(*
SPDX-FileCopyrightText: © 2026 Oleksandr Tiutyk <trofimich@gmail.com>
SPDX-License-Identifier: MIT
License: https://opensource.org/license/mit
*)

{attribute 'no_explicit_call' := 'do not call this function block directly'} 
{attribute 'enable_dynamic_creation'}
FUNCTION_BLOCK WaitAndPickActivity EXTENDS ExclusiveCompositeActivity IMPLEMENTS IWaitAndPickActivity
VAR
	{attribute 'OPC.UA.DA' := '0'}
	_ClassName : STRING := __POUNAME();

	{attribute 'OPC.UA.DA' := '0'}
	_BranchConditions : TOF_Collections.List<0>(0);

	{attribute 'OPC.UA.DA' := '0'}
	_BranchActivities : TOF_Collections.List<0>(0);
	
	{attribute 'OPC.UA.DA' := '0'}	
	_CurrentBranchIndex : DINT := -1;
END_VAR

METHOD AddBarnch : DINT
VAR_INPUT
	condition : ICondition;
	activity : IActivity;
END_VAR
VAR
	conditionNullExcxeption : TOF_Core.ArgumentNotSpecifiedException;
	activityNullExcxeption : TOF_Core.ArgumentNotSpecifiedException;
END_VAR
IF condition = 0  THEN
	activityNullExcxeption.Throw(NamespaceName, ClassName, __POUNAME(), __POSITION(), 'condition');
END_IF

IF activity = 0  THEN
	activityNullExcxeption.Throw(NamespaceName, ClassName, __POUNAME(), __POSITION(), 'activity');
END_IF

activity.ParentActivity := THIS^;

_BranchConditions.AppendGeneric(TOF_Core.GenericValueFactory.FromParts(TOF_Core.GENERIC_TYPE_CLASS.OBJECT, condition.SelfAddress, condition.SelfSize, TOF_Core.GENERIC_MEMORY_MANAGEMENT_BEHAVIOR.STORE_ORIGINAL_REFERENCE_AND_NOT_OWNS_MEMORY));

_BranchActivities.AppendGeneric(TOF_Core.GenericValueFactory.FromParts(TOF_Core.GENERIC_TYPE_CLASS.OBJECT, activity.SelfAddress, activity.SelfSize, TOF_Core.GENERIC_MEMORY_MANAGEMENT_BEHAVIOR.STORE_ORIGINAL_REFERENCE_AND_NOT_OWNS_MEMORY), index => AddBarnch);
END_METHOD

{attribute 'monitoring' := 'call'}
PROPERTY ClassName : REFERENCE TO STRING
GET
ClassName REF= _ClassName;
END_GET
END_PROPERTY

{attribute 'monitoring' := 'call'}
PROPERTY FINAL CurrentActivity : IActivity
GET
IF _BranchActivities.Length > 0 AND_THEN _CurrentBranchIndex >= 0 AND_THEN _CurrentBranchIndex < _BranchActivities.Length THEN
	__QUERYINTERFACE(_BranchActivities.Get(_CurrentBranchIndex).AsObject(), CurrentActivity);
END_IF
END_GET
END_PROPERTY

{attribute 'monitoring' := 'call'}
PROPERTY FINAL CurrentBranchIndex : DINT
GET
CurrentBranchIndex := _CurrentBranchIndex;
END_GET
END_PROPERTY

{attribute 'monitoring' := 'call'}
PROPERTY NamespaceName : REFERENCE TO STRING
GET
NamespaceName REF= CurrentNamespace.Name;
END_GET
END_PROPERTY

METHOD PROTECTED OnCancelling 
VAR_INPUT
	start : BOOL;
END_VAR
VAR_OUTPUT
	cancelled : BOOL;
END_VAR
VAR
	activity : IActivity;
END_VAR
END_METHOD

METHOD PROTECTED OnRunning : ACTIVITY_RUNNING_STATE
VAR_INPUT
	startRunning : BOOL;
	startResuming : BOOL;
END_VAR
VAR_OUTPUT
	haltReason : WSTRING(255);
END_VAR
VAR
	activity : IActivity;
	
	currentActivityNullException : TOF_Core.NullReferenceException;
END_VAR
IF _BranchConditions.Length < 1 THEN
	OnRunning := ACTIVITY_RUNNING_STATE.WORK_COMPLETED;
	RETURN;
END_IF

IF startRunning THEN
	_CurrentBranchIndex := -1;
END_IF

IF _CurrentBranchIndex < 0 THEN
	_CurrentBranchIndex := tryPickBranch();
END_IF

IF _CurrentBranchIndex < 0 THEN
	RETURN;
END_IF

activity := CurrentActivity;

IF activity = 0 THEN
	currentActivityNullException.Throw(NamespaceName, ClassName, __POUNAME(), __POSITION(), 'CurrentActivity');
END_IF

IF startRunning OR_ELSE startResuming OR_ELSE NOT activity.Busy THEN
	activity.RequestStart();
ELSE
	activity.Execute();
END_IF

OnRunning := GetActivityRunningStateByNestedActivityState(activity.State);
END_METHOD

METHOD PROTECTED OnStopping : ACTIVITY_STOPPING_STATE
VAR_INPUT
	startCancelling : BOOL;
	startSuspending : BOOL;
END_VAR
VAR_OUTPUT
	haltReason : WSTRING(255);
END_VAR
VAR
	activity : IActivity;
END_VAR
IF _BranchConditions.Length < 1 THEN
	OnStopping := ACTIVITY_STOPPING_STATE.WORK_COMPLETED;
	RETURN;
END_IF

activity := CurrentActivity;

IF activity = 0 THEN
	IF startCancelling OR_ELSE startSuspending THEN
		OnStopping := ACTIVITY_STOPPING_STATE.WORK_STOPPED;
	ELSE
		OnStopping := ACTIVITY_STOPPING_STATE.WORK_COMPLETED;		
	END_IF

	RETURN;
END_IF

IF NOT activity.Busy THEN
	OnStopping := GetActivityStoppingStateByNestedActivityState(activity.State);
	RETURN;
END_IF

IF startCancelling THEN
	activity.RequestCancel(_CancelReason);
ELSIF startSuspending THEN
	activity.RequestSuspend();
ELSE
	activity.Execute();
END_IF

OnStopping := GetActivityStoppingStateByNestedActivityState(activity.State);
END_METHOD

{attribute 'monitoring' := 'call'}
PROPERTY SelfSize : ULINT
GET
SelfSize := XSIZEOF(THIS^);
END_GET
END_PROPERTY

METHOD PRIVATE tryPickBranch : DINT
VAR
	i : DINT;
	condition : ICondition;
END_VAR
tryPickBranch := -1;

FOR i := 0 TO _BranchConditions.Length - 1 DO
	__QUERYINTERFACE(_BranchConditions.Get(i).AsObject(), condition);
	
	IF condition.Evaluate(THIS^) THEN
		tryPickBranch := i;
		RETURN;
	END_IF
END_FOR
END_METHOD

END_FUNCTION_BLOCK

(* stored: Version 1.1.0.1
   POU WaitAndPickActivity: Id {98b3e546-b646-44e7-bb5b-488f34e41fc2}, SpecialFunc None
   Folder Overriden: Id {85831841-5ba2-46a5-9479-dc90add82035}
   Folder Service members: Id {5438ee75-7621-4c52-a4d9-4dfea8dac7a8}
   Method AddBarnch: Id {f3946fdc-ede0-4f71-bb51-f1411208bc91}
   Property ClassName: Id {0fd055e5-b559-4b38-9ea0-4ca6dfde96f4}
   Get Get: Id {03123722-c59b-4f8b-8e1d-57ef078fc153}
   Property CurrentActivity: Id {ff44d870-a64f-40ed-9ac5-63b06e2e61c2}
   Get Get: Id {8185d1d9-3e50-4bb8-a6f5-2467a7aadc60}
   Property CurrentBranchIndex: Id {33275b8e-2247-47e4-9607-47cd580c7b26}
   Get Get: Id {b77479ef-312c-49a9-8f3c-c0dff4b2b548}
   Property NamespaceName: Id {71b51e02-0e7f-400d-98b6-f6fe9b6e421d}
   Get Get: Id {39b886bb-35c4-4342-9cee-6cf1f6e0a2e1}
   Method OnCancelling: Id {07e9f5dd-2a3d-4db3-89d5-f47d571203f6}
   Method OnRunning: Id {6bdc48e7-942d-42d5-a41d-15bff80339b4}
   Method OnStopping: Id {90584366-9ed4-4c76-823f-f6583e8cb7e4}
   Property SelfSize: Id {f48717c6-b99e-47cb-94a9-c8d92c921628}
   Get Get: Id {2bce559c-e271-4c1b-b7e1-6e1feaa74956}
   Method tryPickBranch: Id {8cf25bf3-94b9-4b19-951a-3c1cbb21bad6} *)
